FUNCTION_BLOCK FB_MoveB EXTENDS FB_StatusExecuteFB
VAR_IN_OUT
	fbMover								: MC_PlanarMover;
END_VAR
VAR_INPUT
	Execute								: BOOL;
	Position							: ST_POSITION;
	Velocity							: LREAL;
	Acceleration						: LREAL;
	Deceleration						: LREAL;
	Jerk								: LREAL;
END_VAR
VAR_OUTPUT
	Done								: BOOL;
	Busy								: BOOL;
	CommandAborted						: BOOL;
	Error								: BOOL;
	ErrorID								: UDINT;
END_VAR
VAR
	uiState								: UINT;
	//Input 内部変数
	dutPosition							: ST_POSITION;
	lrVelocity							: LREAL;
	lrAcceleration						: LREAL;
	lrDeceleration						: LREAL;
	lrJerk								: LREAL;
	
	//ローカル
	fbFB_Mover							: MC_PlanarFeedback;
	fbConstraint						: DynamicConstraint_PathXY;
END_VAR

Prop_Execute := Execute;
METH_Main();

fbFB_Mover.Update();

Busy := bBusy;
Done := bDone;
CommandAborted := bCommandAborted;
Error := bError;
ErrorID := udiErrorID;

//{error 'add method implementation or delete method to use base implementation'}
METHOD INTERNAL METH_Busy : BOOL
{warning disable C0371}
{warning restore C0371}
IF fbFB_Mover.Error THEN
	METH_Error();
	Prop_ErrorID := fbFB_Mover.ErrorId; //Moverがエラー
	RETURN;
END_IF
IF THIS^.fbMover.MCTOPLC.STD.State = MC_PLANAR_STATE.Error THEN
	METH_Error();
	Prop_ErrorID := 1; //Moverがエラー
	RETURN;
END_IF
IF fbFB_Mover.Aborted THEN
	METH_CommandAborted();
	RETURN;
END_IF

CASE THIS^.uiState OF
	0:
	fbConstraint.SetValuesVADJ(V:= THIS^.lrVelocity, A:= THIS^.lrAcceleration, D:= THIS^.lrDeceleration, J:= THIS^.lrJerk);
	THIS^.fbMover.MoveB(
		commandFeedback:= THIS^.fbFB_Mover, 
		targetPosition:= dutPosition.b, 
		constraint:= fbConstraint);

	THIS^.uiState := 10;	
	
	10:
	IF fbFB_Mover.Done THEN
		THIS^.uiState := 16#FFFF;	
	END_IF
	
	16#FFFF:
	METH_Done();
END_CASE
END_METHOD

//{error 'add method implementation or delete method to use base implementation'}
METHOD INTERNAL METH_Enter : BOOL
//Input 内部変数に移す
dutPosition := Position;
lrVelocity := Velocity;
lrAcceleration := Acceleration;
lrDeceleration := Deceleration;
lrJerk := Jerk;
END_METHOD

//{error 'add method implementation or delete method to use base implementation'}
METHOD INTERNAL METH_Exit : BOOL
Prop_Done := FALSE;
Prop_Busy := FALSE;
Prop_CommandAborted := FALSE;
Prop_Error := FALSE;
Prop_ErrorID := 0;

// 内部変数をリフレッシュする
uiState := 0;
lrVelocity := 0;
lrAcceleration := 0;
lrDeceleration := 0;
lrJerk := 0;
END_METHOD

//{error 'add method implementation or delete method to use base implementation'}
METHOD INTERNAL METH_Main : BOOL
//Doneに遷移
IF SUPER^.bDone AND SUPER^.bExecute THEN
	METH_Done();
	RETURN;
END_IF
//Errorに遷移
IF SUPER^.bError AND SUPER^.bExecute THEN
	METH_Error();
	RETURN;
END_IF
//CommandAbortedに遷移
IF SUPER^.bCommandAborted AND SUPER^.bExecute THEN
	METH_CommandAborted();
	RETURN;
END_IF
//FBをリフレッシュ
//状態がDone, Error, CommandAborted時に Execute FALSE で遷移
IF (SUPER^.bDone OR SUPER^.bError OR SUPER^.bCommandAborted) AND NOT SUPER^.bExecute THEN
	METH_Exit();
	RETURN;
END_IF

//実行開始
IF SUPER^.bExecute AND NOT SUPER^.bBusy THEN
	METH_Execute();
	METH_Enter();
END_IF
//実行中
IF SUPER^.bBusy THEN
	METH_Busy();
END_IF
END_METHOD

END_FUNCTION_BLOCK

(* stored: Version 1.1.0.1, ProductVersion 3.1.4024.12
   POU FB_MoveB: Id {8425ca0d-2577-471e-a0ef-1098251f657b}, SpecialFunc None
   Method METH_Busy: Id {79f51cc3-e95a-4bad-b4da-50ca607e8601}
   Method METH_Enter: Id {5f9a41b4-098b-488f-85ba-b8a5895db5db}
   Method METH_Exit: Id {21f5cad7-bd12-4237-814d-ed0257c8e35b}
   Method METH_Main: Id {f09c1c56-7ade-4a5a-abdb-2c9c86a841e5} *)
